// TIA Portal project "YouTube" (V15.1)

(* hardware
DEVICE "S71500/ET200MP station_1"  S7-1500 station
   slot 0: "Rail_0"  Rack  6ES7 590-1***0-0AA0
   slot 1: "Brain"  CPU 1512C-1 PN  6ES7 512-1CK00-0AB0  V1.8
      slot 3: "CPU display_1"  6ES7591-1AA00-0AA0
   slot 2: "DI 16x24VDC / DQ 16x24VDC/0.5A BA_1"  DI 16/DQ 16x24VDC  6ES7 523-1BL00-0AA0  V1.0
*)

// ===== PLC "Brain"  CPU 1512C-1 PN =====

VAR_GLOBAL   // PLC tag table "Default tag table"
   "Tag_1" AT %M1.1 : Bool;
END_VAR

VAR_GLOBAL   // PLC tag table "Inputs and Outputs"
   "K1" AT %Q4.0 : Bool;   // Onveyr Belt on
   "1M1" AT %Q4.1 : Bool;   // Open stopper
   "B1" AT %I10.0 : Bool;   // Component at conveyr start
   "B2" AT %I10.1 : Bool;   // Componenet at conveyr center
   "B3" AT %I10.2 : Bool;   // No Componenet at conveyr
   "S1" AT %I10.3 : Bool;   // Start button
   "P1" AT %Q4.2 : Bool;   // Indicator LED
   "B20" AT %I10.4 : Bool;   // Color detection
   "K1.1" AT %Q4.3 : Bool;   // Conveyr Belt reverse
END_VAR

VAR_GLOBAL   // PLC tag table "Clock memory"
   "Clock_Byte" AT %MB0 : Byte;
   "Clock_10Hz" AT %M0.0 : Bool;
   "Clock_5Hz" AT %M0.1 : Bool;
   "Clock_2.5Hz" AT %M0.2 : Bool;
   "Clock_2Hz" AT %M0.3 : Bool;
   "Clock_1.25Hz" AT %M0.4 : Bool;
   "Clock_1Hz" AT %M0.5 : Bool;
   "Clock_0.625Hz" AT %M0.6 : Bool;
   "Clock_0.5Hz" AT %M0.7 : Bool;
END_VAR

DATA_BLOCK "Conveyr Sequence_DB"   // DB1
{ S7_Optimized_Access := 'TRUE' }
VERSION : 0.1
// stored: InstanceOfName Conveyr Sequence
"Conveyr Sequence"
BEGIN
END_DATA_BLOCK

FUNCTION_BLOCK "Conveyr Sequence"   // FB1, GRAPH_PLUS
{ S7_Optimized_Access := 'TRUE' }
VERSION : 0.1
   VAR_INPUT
      OFF_SQ : Bool := false;   // Turn sequence off
      INIT_SQ : Bool := false;   // Set sequence to initial state
      ACK_EF : Bool := false;   // Acknowledge all errors and faults
      S_PREV : Bool := false;   // Output previous step in parameter S_NO
      S_NEXT : Bool := false;   // Indicate next step in parameter S_NO
      SW_AUTO : Bool := false;   // Automatic mode
      SW_TAP : Bool := false;   // Semiautomatic/switch with transition
      SW_TOP : Bool := false;   // Semiautomatic/ignore transition
      SW_MAN : Bool := false;   // Manual mode
      S_SEL : Int := 0;   // Select step to be output to S_NO
      S_ON : Bool := false;   // Activate step indicated in S_NO
      S_OFF : Bool := false;   // Deactivate step indicated S_NO
      T_PUSH : Bool := false;   // Enable transition to switch in semi automatic mode
   END_VAR
   VAR_OUTPUT
      S_NO : Int := 0;   // Step number
      S_MORE : Bool := false;   // More steps are available and can be shown in S_NO
      S_ACTIVE : Bool := false;   // Step indicated in S_NO is active
      ERR_FLT : Bool := false;   // Interlock or supervision group error
      AUTO_ON : Bool := false;   // Automatic mode is active
      TAP_ON : Bool := false;   // Semiautomatic mode/step with transition enabled
      TOP_ON : Bool := false;   // Semiautomatic mode/ignore transition enabled
      MAN_ON : Bool := false;   // Manual mode is active
   END_VAR
   VAR
      HMI_INFO : Array[0..8] of UInt;
      IF_PAR : G7_IfParPlus_V2;
      RT_DATA : G7_RTDataPlus_V2;   // Internal data area
      "Waiting  for Peace" : G7_TransitionPlus_V2;   // Transition structure
      "In Center posotion" : G7_TransitionPlus_V2;   // Transition structure
      "Not In Center" : G7_TransitionPlus_V2;   // Transition structure
      "In End Position" : G7_TransitionPlus_V2;   // Transition structure
      "Belt Empty" : G7_TransitionPlus_V2;   // Transition structure
      "Itinial Step" : G7_StepPlus_V2;   // Step structure
      "Start Conveyr" : G7_StepPlus_V2;   // Step structure
      "Open Stopper" : G7_StepPlus_V2;   // Step structure
      "Continue Conveyr" : G7_StepPlus_V2;   // Step structure
      "Wait for empty belt" : G7_StepPlus_V2;   // Step structure
      SINI : Array[0..1] of USInt;
      LSTT : Array[0..4] of USInt;
      ATAJ : Array[0..4] of USInt;
      ATAB : Array[0..4] of USInt;
      PSTT : Array[0..4] of USInt;
      NSTT : Array[0..4] of USInt;
      ASSJ : Array[0..4] of USInt;
      ASSB : Array[0..4] of USInt;
      PTTS : Array[0..4] of USInt;
      NTTS : Array[0..4] of USInt;
      SW_SQTS : Array[0..4] of USInt;
      SWITCH : Array[0..0] of USInt;
      TVX : Array[0..1] of USInt;
      TTX : Array[0..1] of USInt;
      TSX : Array[0..1] of USInt;
      S00X : Array[0..1] of USInt;
      SOFFX : Array[0..1] of USInt;
      SONX : Array[0..1] of USInt;
      SAX : Array[0..1] of USInt;
      SERRX : Array[0..5] of USInt;
      SMX : Array[0..5] of USInt;
      S0X : Array[0..5] of USInt;
      S1X : Array[0..5] of USInt;
      IL_ALARM_INST : Program_Alarm;
      SUP_ALARM_INST : Program_Alarm;
      STEP_TIME_ALARM_INST : Program_Alarm;
      IEC_TIMER_INST : IEC_TIMER;
      TRANSACTION_FLAG : Bool := false;
      "In Center grey part" : G7_TransitionPlus_V2;   // Transition structure
      "Conveyr Reverse" : G7_StepPlus_V2;   // Step structure
      "Back At Start" : G7_TransitionPlus_V2;   // Transition structure
      "Wait for empty" : G7_StepPlus_V2;   // Step structure
      Trans8 : G7_TransitionPlus_V2;   // Transition structure
   END_VAR
   // SINI[0] := 2;
   // LSTT[0] := 255;
   // LSTT[1] := 255;
   // LSTT[2] := 255;
   // LSTT[3] := 255;
   // ATAJ[1] := 1;
   // ATAJ[2] := 2;
   // ATAJ[3] := 3;
   // ATAJ[4] := 4;
   // ATAB[1] := 1;
   // ATAB[2] := 2;
   // ATAB[3] := 3;
   // ATAB[4] := 4;
   // PSTT[1] := 1;
   // PSTT[2] := 2;
   // PSTT[3] := 3;
   // PSTT[4] := 4;
   // NSTT[0] := 1;
   // NSTT[1] := 2;
   // NSTT[2] := 3;
   // NSTT[3] := 4;
   // ASSJ[1] := 1;
   // ASSJ[2] := 2;
   // ASSJ[3] := 3;
   // ASSJ[4] := 4;
   // ASSB[1] := 1;
   // ASSB[2] := 2;
   // ASSB[3] := 3;
   // ASSB[4] := 4;
   // PTTS[0] := 255;
   // PTTS[2] := 1;
   // PTTS[3] := 2;
   // PTTS[4] := 3;
   // NTTS[1] := 1;
   // NTTS[2] := 2;
   // NTTS[3] := 3;
   // NTTS[4] := 4;
   // TVX[0] := 16#1;
   // TTX[0] := 16#1;
   // TSX[0] := 16#1;
   // S00X[0] := 16#1;
   // SOFFX[0] := 16#1;
   // SONX[0] := 16#1;
   // SAX[0] := 16#1;
   // SERRX[0] := 16#1;
   // SMX[0] := 16#1;
   // S0X[0] := 16#1;
   // S1X[0] := 16#1;
BEGIN
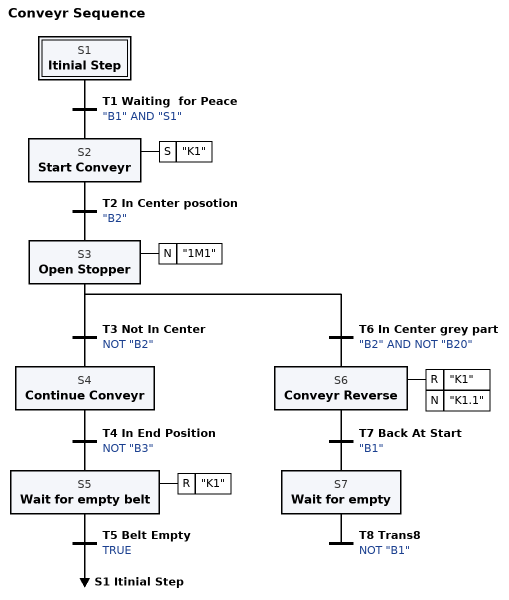
   // sequencer 1
   INITIAL_STEP "Itinial Step":   // S1, max time T#10S, warning time T#7S
   END_STEP
   TRANSITION "Waiting  for Peace" FROM "Itinial Step" TO "Start Conveyr"   // T1
      := "B1" AND "S1";
   END_TRANSITION
   STEP "Start Conveyr":   // S2, max time T#10S, warning time T#7S
              S    "K1"
   END_STEP
   TRANSITION "In Center posotion" FROM "Start Conveyr" TO "Open Stopper"   // T2
      := "B2";
   END_TRANSITION
   STEP "Open Stopper":   // S3, max time T#10S, warning time T#7S
              N    "1M1"
   END_STEP
   TRANSITION "Not In Center" FROM "Open Stopper" TO "Continue Conveyr"   // T3
      := NOT "B2";
   END_TRANSITION
   TRANSITION "In Center grey part" FROM "Open Stopper" TO "Conveyr Reverse"   // T6
      := "B2" AND NOT "B20";
   END_TRANSITION
   STEP "Continue Conveyr":   // S4, max time T#10S, warning time T#7S
   END_STEP
   TRANSITION "In End Position" FROM "Continue Conveyr" TO "Wait for empty belt"   // T4
      := NOT "B3";
   END_TRANSITION
   STEP "Wait for empty belt":   // S5, max time T#10S, warning time T#7S
              R    "K1"
   END_STEP
   TRANSITION "Belt Empty" FROM "Wait for empty belt" TO "Itinial Step"   // T5, jump
      := TRUE;
   END_TRANSITION
   STEP "Conveyr Reverse":   // S6, max time T#10S, warning time T#7S
              R    "K1"
              N    "K1.1"
   END_STEP
   TRANSITION "Back At Start" FROM "Conveyr Reverse" TO "Wait for empty"   // T7
      := "B1";
   END_TRANSITION
   STEP "Wait for empty":   // S7, max time T#10S, warning time T#7S
   END_STEP
   TRANSITION Trans8 FROM "Wait for empty" TO ?   // T8
      := NOT "B1";
   END_TRANSITION
END_FUNCTION_BLOCK

FUNCTION "Conveyr" : Void   // FC1, LAD
{ S7_Optimized_Access := 'TRUE' }
VERSION : 0.1
   VAR_INPUT
      "Conveyr Start" : Bool;
      "Conveyr Center" : Bool;
      "Conveyr End" : Bool;
      "Start Button" : Bool;
      "Conveyr On Frequency" : Bool;
      "Part at Start Frequency" : Bool;
   END_VAR
   VAR_OUTPUT
      Stopper : Bool;
      LED : Bool;
   END_VAR
   VAR_IN_OUT
      Conveyr : Bool;
   END_VAR
BEGIN

REGION Network 1
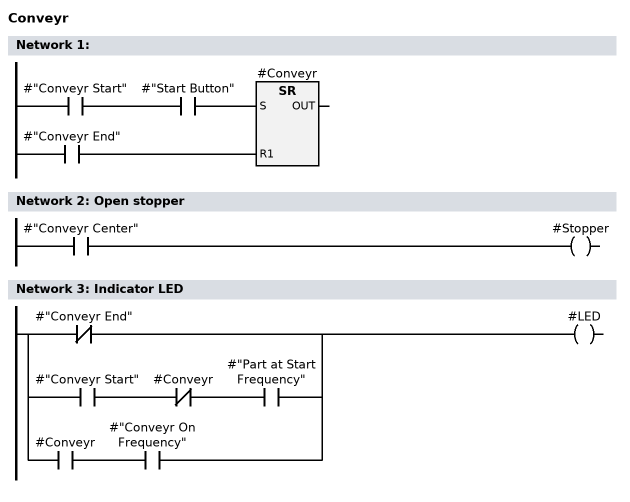
   RUNG wire#powerrail
      Contact( #"Conveyr Start" )
      Contact( #"Start Button" )
      S_SR(operand := #Conveyr, r1 := wire#w1)
   END_RUNG
   RUNG wire#powerrail
      Contact( #"Conveyr End" )
   END_RUNG wire#w1
   // the same network as SCL:
   IF #"Conveyr Start" AND #"Start Button" THEN
       #Conveyr := TRUE;   // SR flip-flop
   END_IF;
   IF #"Conveyr End" THEN #Conveyr := FALSE; END_IF;
END_REGION

REGION Network 2: Open stopper
   RUNG wire#powerrail
      Contact( #"Conveyr Center" )
      Coil( #Stopper )
   END_RUNG
   // the same network as SCL:
   #Stopper := #"Conveyr Center";
END_REGION

REGION Network 3: Indicator LED
   RUNG wire#powerrail
      I_Contact( #"Conveyr End" )
      wire#w1
      Coil( #LED )
   END_RUNG
   RUNG wire#powerrail
      Contact( #"Conveyr Start" )
      I_Contact( #Conveyr )
      Contact( #"Part at Start Frequency" )
   END_RUNG wire#w1
   RUNG wire#powerrail
      Contact( #Conveyr )
      Contact( #"Conveyr On Frequency" )
   END_RUNG wire#w1
   // the same network as SCL:
   #LED := NOT #"Conveyr End" OR (#"Conveyr Start" AND NOT #Conveyr AND #"Part at Start Frequency") OR (#Conveyr AND #"Conveyr On Frequency");
END_REGION
END_FUNCTION

ORGANIZATION_BLOCK "Main"   // OB1, LAD, ProgramCycle
TITLE = "Main Program Sweep (Cycle)"
{ S7_Optimized_Access := 'TRUE' }
VERSION : 0.1
   VAR_INPUT
      Initial_Call : Bool;   // Initial call of this OB
      Remanence : Bool;   // =True, if remanent data are available
   END_VAR
BEGIN

REGION Network 1
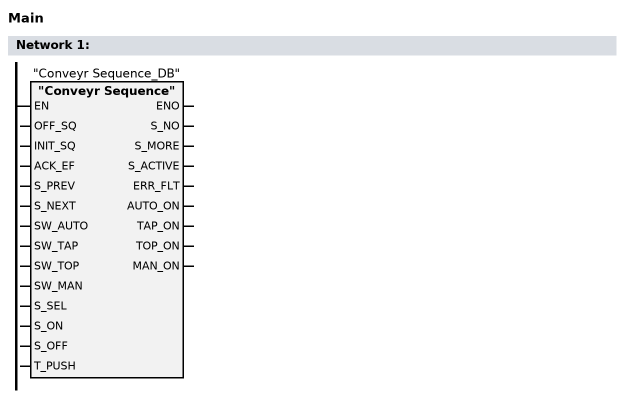
   RUNG wire#powerrail
      "Conveyr Sequence_DB"(OFF_SQ :=, INIT_SQ :=, ACK_EF :=, S_PREV :=, S_NEXT :=, SW_AUTO :=, SW_TAP :=, SW_TOP :=, SW_MAN :=, S_SEL :=, S_ON :=, S_OFF :=, T_PUSH :=, S_NO =>, S_MORE =>, S_ACTIVE =>, ERR_FLT =>, AUTO_ON =>, TAP_ON =>, TOP_ON =>, MAN_ON =>)
   END_RUNG
   // the same network as SCL:
   "Conveyr Sequence_DB"();   // "Conveyr Sequence"
END_REGION
END_ORGANIZATION_BLOCK